{attribute 'no_check'}
FUNCTION_BLOCK AnalogOut_EL2535 EXTENDS AnalogOut
VAR_INPUT
	Reset										AT  %Q*		:	BOOL;	
END_VAR   
VAR_IN_OUT
END_VAR              									                              	            	
VAR_OUTPUT                              	            	
	Input										AT  %I* 	: 	BOOL; 	//Hardware Input 
	ReadyToEnable								AT  %I* 	: 	BOOL; 	
	Warning										AT  %I* 	: 	BOOL; 	
	Error										AT  %I* 	: 	BOOL; 	
	TxPDOToggle									AT  %I* 	: 	BOOL; 	
            
	InfoData1									AT  %I* 	: 	INT; //Actual current
	InfoData2									AT  %I* 	: 	INT; //Duty cycle/Voltage
END_VAR                                 	
VAR                                     	
END_VAR

(* Set PWM Output of EL25xx																					*)
(************************************************************************************************************)
	SUPER^();

(********************************************************************************************************)

END_FUNCTION_BLOCK

(* stored: Version 1.1.0.1, ProductVersion 3.1.4024.13
   POU AnalogOut_EL2535: Id {aca08393-a9c7-4de5-b6d8-5e739d8aca09}, SpecialFunc None *)
